{attribute 'linkalways'} 
{attribute 'no_explicit_call' := 'This FB is a CLASS and must be accessed using methods or properties'}
{attribute 'enable_dynamic_creation'}
FUNCTION_BLOCK _ETcVnFeatureScalingType EXTENDS EnumDatatypeBase
VAR
	localData : ETcVnFeatureScalingType;
	activeData : REFERENCE TO ETcVnFeatureScalingType;
	enumBaseDatatype : _DINT(localData);
END_VAR

METHOD PRIVATE AddLocalEnumeration
VAR_INPUT
	Enumeration : T_MAXSTRING;
	Value : ETcVnFeatureScalingType;
END_VAR
AddEnumeration(Enumeration, Value);
END_METHOD

PROPERTY PUBLIC Address : PVOID
GET
Address := ADR(activeData);
END_GET
END_PROPERTY

METHOD PUBLIC ClearReference
VAR_INPUT
END_VAR
activeData REF= localData;
SetBaseDatatypeReference();
END_METHOD

METHOD PUBLIC Clone : I_Datatype
VAR
    pClone : POINTER TO _ETcVnFeatureScalingType;
END_VAR
pClone := __NEW(_ETcVnFeatureScalingType(InitialValue := Value));
Clone := pClone^;
END_METHOD

METHOD FB_init : BOOL
VAR_INPUT
	bInitRetains : BOOL; // if TRUE, the retain variables are initialized (warm start / cold start)
	bInCopyCode : BOOL;  // if TRUE, the instance afterwards gets moved into the copy code (online change)
	InitialValue : ETcVnFeatureScalingType;
END_VAR
localData := InitialValue;
AddBaseDatatype(enumBaseDatatype);
ClearReference();

AddLocalEnumeration('TCVN_FST1_MAXABS', ETcVnFeatureScalingType.TCVN_FST1_MAXABS);
AddLocalEnumeration('TCVN_FST1_MINMAX', ETcVnFeatureScalingType.TCVN_FST1_MINMAX);
AddLocalEnumeration('TCVN_FST1_STANDARDIZATION', ETcVnFeatureScalingType.TCVN_FST1_STANDARDIZATION);
END_METHOD

PROPERTY PUBLIC Identifier : T_MAXSTRING
GET
Identifier := 'ETcVnFeatureScalingType';
END_GET
END_PROPERTY

METHOD IsEnumeratorValueEqual : BOOL
VAR_INPUT
	Enumerator : I_KeyValueForwardEnumerator;
END_VAR
VAR
	storedValue : ETcVnFeatureScalingType;
END_VAR
IF NOT Enumerator.TryGet(storedValue) THEN
	RETURN;
END_IF

IsEnumeratorValueEqual := storedValue = activeData;
END_METHOD

METHOD PUBLIC MakeReferenceTo
VAR_INPUT
	ReferenceTarget : REFERENCE TO ETcVnFeatureScalingType;
END_VAR
activeData REF= ReferenceTarget;
SetBaseDatatypeReference();
END_METHOD

METHOD PROTECTED SetBaseDatatypeReference
VAR_INPUT
END_VAR
enumBaseDatatype.MakeReferenceTo(activeData);
END_METHOD

PROPERTY PUBLIC Size : UDINT
GET
Size := SIZEOF(activeData);
END_GET
END_PROPERTY

METHOD TryMakeReferenceTo : BOOL
VAR_INPUT
	Target : I_Datatype;
END_VAR
VAR
	targetAsEnum : I_EnumDatatype;
	pTargetData : POINTER TO ETcVnFeatureScalingType;
END_VAR
IF NOT Target.TryResolveAsEnumDatatype(targetAsEnum) THEN
	RETURN;
END_IF

IF targetAsEnum.Identifier <> Identifier THEN
	RETURN;
END_IF

pTargetData := Target.Address;
activeData REF= pTargetData^;
SetBaseDatatypeReference();
TryMakeReferenceTo := TRUE;
END_METHOD

PROPERTY PUBLIC Value : ETcVnFeatureScalingType
GET
Value := activeData;
END_GET
SET
activeData := Value;
END_SET
END_PROPERTY

END_FUNCTION_BLOCK

(* stored: Version 1.1.0.1, ProductVersion 3.1.4024.12
   POU _ETcVnFeatureScalingType: Id {ead42140-2b39-4a15-ac16-2be66e0d4a44}, SpecialFunc None
   Folder Constructor: Id {e67468ce-3486-4f09-afe0-a47c881ce9b8}
   Folder Private: Id {3a030e10-2915-4412-ac94-cff591fea235}
   Folder Protected: Id {5b98c273-07f0-4dea-9926-e05ba0c8c980}
   Method AddLocalEnumeration: Id {83ea937b-77b2-4553-9b28-62381dbce3ad}
   Property Address: Id {f133f592-93ec-4188-8eb6-04a44d53d2eb}
   Get Get: Id {244ee61e-9a8f-44f3-b28b-ac3bc842dae3}
   Method ClearReference: Id {2346c4ee-65b9-4245-aee6-868303f38728}
   Method Clone: Id {4043b563-ef98-4d10-988e-8f0286d7b66b}
   Method FB_init: Id {8b7dcae6-72a7-4d87-b3f9-8bd60ac1f1c2}
   Property Identifier: Id {862c136f-6ca6-4083-ae23-0bb152c07f5f}
   Get Get: Id {ae98170d-31e7-4f31-a2cd-b9bd1ca9c6b3}
   Method IsEnumeratorValueEqual: Id {3279d032-cfc0-4e6a-91d5-31bce04a1540}
   Method MakeReferenceTo: Id {767d244f-11cf-4828-a66f-fa68fc8d6d8b}
   Method SetBaseDatatypeReference: Id {b3da4ce2-9d26-4ca3-b1e7-efc8ab5151f9}
   Property Size: Id {d2643df7-d3c0-4e74-ad9f-83ae260b04d0}
   Get Get: Id {c96b9e50-584d-4dc9-a200-28b5098746b2}
   Method TryMakeReferenceTo: Id {ec1ae0e1-f073-47db-9404-71a8449fc54e}
   Property Value: Id {2a7d815f-77de-4a40-9917-de2561ed1af4}
   Get Get: Id {b7a50e27-0529-4099-bd2d-7a517a34ff17}
   Set Set: Id {86afa9a6-4fb9-4e77-a99f-62a4950962e5} *)
